TYPE T_AnyIntOrBit : __SYSTEM.AnyType; END_TYPE

(* stored: Version 1.1.0.1
   DUT T_AnyIntOrBit: Id {e2f912fc-26e3-4cc2-87bd-76e1078e50ef} *)
